FUNCTION_BLOCK FB_MqttCoverPositionDiscovery EXTENDS FB_MqttDeviceDiscoveryBase
VAR_INPUT
END_VAR
VAR_OUTPUT
END_VAR
VAR
	stConfig : ST_MqttCoverPositionConfiguration;
END_VAR

PROPERTY PROTECTED Component : STRING(30)
GET
Component := 'cover';
END_GET
END_PROPERTY

METHOD  ConfigToJson : STRING(1000)
VAR_INPUT
END_VAR
VAR
	fbJsonWriter : FB_JsonSaxWriter;
END_VAR
fbJsonWriter.ResetDocument();
fbJsonWriter.StartObject();
fbJsonWriter.AddKeyString(key := 'cmd_t', value := THIS^.stConfig.command_topic);
fbJsonWriter.AddKeyString(key := 'pos_t', value := THIS^.stConfig.position_topic);
fbJsonWriter.AddKeyString(key := 'set_pos_t', value := THIS^.stConfig.set_position_topic);
fbJsonWriter.AddKeyString(key := 'pl_open', value := THIS^.stConfig.payload_open);
fbJsonWriter.AddKeyString(key := 'pl_cls', value := THIS^.stConfig.payload_close);
fbJsonWriter.AddKeyString(key := 'pl_stop', value := THIS^.stConfig.payload_stop);
fbJsonWriter.AddKeyNumber(key := 'pos_open', value := THIS^.stConfig.position_open);
fbJsonWriter.AddKeyNumber(key := 'pos_clsd', value := THIS^.stConfig.position_closed);
fbJsonWriter.AddKeyString(key := 'dev_cla', value := THIS^.stConfig.device_class);
fbJsonWriter.AddKeyBool(key := 'opt', value := THIS^.stConfig.optimistic);
fbJsonWriter.AddKeyString(key := 'uniq_id', value := THIS^.stConfig.unique_id);
fbJsonWriter.AddKeyString(key := 'name', value := this^.stConfig.name);
THIS^.DevInfoToJson(rJsonWriter := fbJsonWriter);
fbJsonWriter.EndObject();
fbJsonWriter.CopyDocument(pDoc := ConfigToJson, nDoc := 1000);
END_METHOD

PROPERTY Configuration : ST_MqttCoverPositionConfiguration
GET
Configuration := this^.stConfig;
END_GET
SET
this^.stConfig := Configuration;
END_SET
END_PROPERTY

END_FUNCTION_BLOCK

(* stored: Version 1.1.0.1, ProductVersion 3.1.4024.5
   POU FB_MqttCoverPositionDiscovery: Id {8f1e903a-7212-45ea-81b6-d4e9a543b138}, SpecialFunc None
   Property Component: Id {c29211bf-77a2-41ef-9e16-76709f71f284}
   Get Get: Id {fcb74905-6479-4318-b959-0ee8dc1cb7c9}
   Method ConfigToJson: Id {4bc9cc79-fcbc-464c-94c2-fcd98d0296a0}
   Property Configuration: Id {8ea59188-aa41-4db8-896e-0d19078e52d4}
   Get Get: Id {e1d24410-0f53-4811-bb3e-45251393877f}
   Set Set: Id {ac1bc800-5016-4ed7-b3ba-18cc265964f5} *)
